FUNCTION_BLOCK mySimpleBlock (* Simple FB with one algorithm *)
  (* Standard: 61499-1 *)
  (* Version 1.0, 2025-07-10, dakudryashev *)
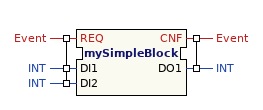
  EVENT_INPUT
    REQ WITH DI1, DI2; (* Normal Execution Request *)
  END_EVENT
  EVENT_OUTPUT
    CNF WITH DO1; (* Execution Confirmation *)
  END_EVENT
  VAR_INPUT
    DI1 : INT;
    DI2 : INT;
  END_VAR
  VAR_OUTPUT
    DO1 : INT;
  END_VAR
  EC_STATES
    REQ : REQ -> CNF;
  END_STATES
  ALGORITHM REQ IN ST:
DO1 := DI1 + DI2;
  END_ALGORITHM
END_FUNCTION_BLOCK
